FUNCTION FC_MemcpyLimited : BOOL
VAR_INPUT
	DestinationAdress			: PVOID;
	ediSizeOfDestAdress			: UDINT;
	
	SourceAdress				: PVOID;
	ediBytesToCopy				: UDINT;
END_VAR
VAR
	tdiBytesToCopy				: UDINT;
END_VAR

tdiBytesToCopy := LIMIT(0, ediBytesToCopy, ediSizeOfDestAdress);

MEMCPY(DestinationAdress, SourceAdress, tdiBytesToCopy);

END_FUNCTION

(* stored: Version 1.1.0.1, ProductVersion 3.1.4024.12
   POU FC_MemcpyLimited: Id {e30c5c0b-ae61-4333-8eaa-a16b9553d76c}, SpecialFunc None *)
